// TIA Portal V16 export
// export: Created 2022-07-21T09:35:31.3683983Z, ExportSetting WithDefaults, DisplayName Totally Integrated Automation Portal, DisplayVersion V16 Update 4, DisplayName TIA Portal Version Control Interface, DisplayVersion V16 Update 2, DisplayName TIA Portal Openness, DisplayVersion V16 Update 4, DisplayName SINAMICS Startdrive Advanced, DisplayVersion V16 Update 5, DisplayName SINAMICS Startdrive G130, G150, S120, S150, SINAMICS MV, S210, DisplayVersion V16 Update 5, DisplayName SINAMICS Startdrive G110M, G120, G120C, G120D, G120P, G115D, DisplayVersion V16 Update 5, DisplayName STEP 7 Professional, DisplayVersion V16 Update 4, DisplayName STEP 7 Safety, DisplayVersion V16, DisplayName WinCC Advanced, DisplayVersion V16 Update 4
FUNCTION "fcCommand" : Void   // FC11, LAD
TITLE = Output handling / Obsługa wyjść
{ S7_Optimized_Access := 'TRUE' }
VERSION : 0.1
// stored: AutoNumber true, IsIECCheckEnabled false, SetENOAutomatically false, UDAEnableTagReadback false
   VAR_INPUT
      inResetEnergySaving : Bool;
      inStopImediatelly : Bool;
      inError : Bool;
   END_VAR
   VAR_OUTPUT
      ouCommand : "typeCommand";
   END_VAR
BEGIN

REGION Network 1: Copy inputs to outputs / Przepisanie wejść na wyjścia
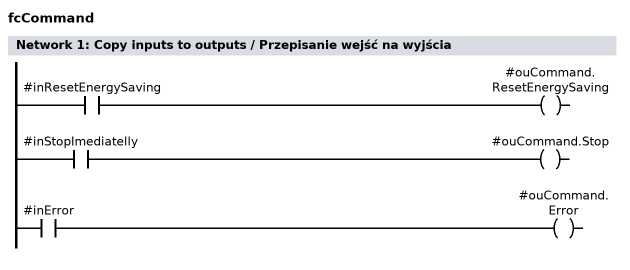
   RUNG wire#powerrail
      Contact( #inResetEnergySaving )
      Coil( #ouCommand.ResetEnergySaving )
   END_RUNG
   RUNG wire#powerrail
      Contact( #inStopImediatelly )
      Coil( #ouCommand.Stop )
   END_RUNG
   RUNG wire#powerrail
      Contact( #inError )
      Coil( #ouCommand.Error )
   END_RUNG
   // the same network as SCL:
   #ouCommand.ResetEnergySaving := #inResetEnergySaving;
   #ouCommand.Stop := #inStopImediatelly;
   #ouCommand.Error := #inError;
END_REGION
END_FUNCTION
